PROGRAM LASER_PROG
VAR
	
	PULS1: TON;
	PULS2: TON;
	CNT1: CTU;
	LOTBOX_ACC: INT;
	LOTBOX_ACC1: INT;
	LOTBOX_TEMP1: INT;
	LOTBOX_TEMP2: INT;
	LOTBOX_TEMP3: INT;
	LOTBOX_TEMP4: INT;
	NGBOX_TEMP: INT;
	NGBOX_TEMP1: INT;
	NGBOX_TEMP2: INT;
	NGBOX_TEMP3: INT;
	NGBOX_TEMP4: INT;
	NGBOX_ACC: INT;
END_VAR


PULS1(IN:=NOT PULS2.Q,PT:=T#0.5S);
PULS2(IN:=PULS1.Q,PT:=T#1S);
CNT1(CU:=PULS1.Q,RESET:=CNT1.Q,PV:=9);
(*
IF CNT1.CV=1 THEN
	SORTER_VAR.O_NG_BOX_INDICATOR_4:=TRUE;
END_IF
IF CNT1.CV=2 THEN
	SORTER_VAR.O_NG_BOX_INDICATOR_3:=TRUE;
END_IF
IF CNT1.CV=3 THEN
	SORTER_VAR.O_NG_BOX_INDICATOR_2:=TRUE;
END_IF
IF CNT1.CV=4 THEN
	SORTER_VAR.O_NG_BOX_INDICATOR_1:=TRUE;
END_IF
IF CNT1.CV=5 THEN
	SORTER_VAR.O_LOT_BOX_INDICATOR_4:=TRUE;
END_IF
IF CNT1.CV=6 THEN
	SORTER_VAR.O_LOT_BOX_INDICATOR_3:=TRUE;
END_IF
IF CNT1.CV=7 THEN
	SORTER_VAR.O_LOT_BOX_INDICATOR_2:=TRUE;
END_IF
IF CNT1.CV=8 THEN
	SORTER_VAR.O_LOT_BOX_INDICATOR_1:=TRUE;
END_IF
IF CNT1.Q THEN
	SORTER_VAR.O_LOT_BOX_INDICATOR_1:=FALSE;
	SORTER_VAR.O_LOT_BOX_INDICATOR_2:=FALSE;
	SORTER_VAR.O_LOT_BOX_INDICATOR_3:=FALSE;
	SORTER_VAR.O_LOT_BOX_INDICATOR_4:=FALSE;
	SORTER_VAR.O_NG_BOX_INDICATOR_1:=FALSE;
	SORTER_VAR.O_NG_BOX_INDICATOR_2:=FALSE;
	SORTER_VAR.O_NG_BOX_INDICATOR_3:=FALSE;
	SORTER_VAR.O_NG_BOX_INDICATOR_4:=FALSE;
END_IF
*)
IF SORTER_VAR.I_LOTBOX_DETECT_1 THEN
	SORTER_VAR.O_LOT_BOX_INDICATOR_1:=PULS1.Q;
	LOTBOX_TEMP1:=1;
ELSE
	SORTER_VAR.O_LOT_BOX_INDICATOR_1:=FALSE;
	LOTBOX_TEMP1:=0;
END_IF

IF SORTER_VAR.I_LOTBOX_DETECT_2 THEN
	SORTER_VAR.O_LOT_BOX_INDICATOR_2:=PULS1.Q;
	LOTBOX_TEMP2:=1;
	ELSE
	LOTBOX_TEMP2:=0;
	SORTER_VAR.O_LOT_BOX_INDICATOR_2:=FALSE;
END_IF

IF SORTER_VAR.I_LOTBOX_DETECT_3 THEN
	SORTER_VAR.O_LOT_BOX_INDICATOR_3:=PULS1.Q;
	LOTBOX_TEMP3:=1;
	ELSE
	SORTER_VAR.O_LOT_BOX_INDICATOR_3:=FALSE;
	LOTBOX_TEMP3:=0;
END_IF

IF SORTER_VAR.I_LOTBOX_DETECT_4 THEN
	SORTER_VAR.O_LOT_BOX_INDICATOR_4:=PULS1.Q;
	LOTBOX_TEMP4:=1;
	ELSE
	SORTER_VAR.O_LOT_BOX_INDICATOR_4:=FALSE;
	LOTBOX_TEMP4:=0;
END_IF
LOTBOX_ACC:=LOTBOX_TEMP1 +LOTBOX_TEMP2+LOTBOX_TEMP3+LOTBOX_TEMP4;

IF LOTBOX_ACC >=3 THEN
	//SORTER_VAR.O_TOWER_LAMP_BUZZER :=TRUE;
	ELSE
	SORTER_VAR.O_TOWER_LAMP_BUZZER :=FALSE;
END_IF

IF NOT SORTER_VAR.I_NG_BOX_DETECT_1 THEN
		SORTER_VAR.O_NG_BOX_INDICATOR_1:=PULS1.Q;
		NGBOX_TEMP1:=1;
		ELSE
		SORTER_VAR.O_NG_BOX_INDICATOR_1:=FALSE;
		NGBOX_TEMP1:=0;
END_IF

IF NOT SORTER_VAR.I_NG_BOX_DETECT_2 THEN
		SORTER_VAR.O_NG_BOX_INDICATOR_2:=PULS1.Q;
		NGBOX_TEMP2:=1;
		ELSE
		SORTER_VAR.O_NG_BOX_INDICATOR_2:=FALSE;
		NGBOX_TEMP2:=0;
END_IF

IF NOT SORTER_VAR.I_NG_BOX_DETECT_3 THEN
		SORTER_VAR.O_NG_BOX_INDICATOR_3:=PULS1.Q;
		NGBOX_TEMP3:=1;
		ELSE
		SORTER_VAR.O_NG_BOX_INDICATOR_3:=FALSE;
		NGBOX_TEMP3:=0;
END_IF

IF NOT SORTER_VAR.I_NG_BOX_DETECT_4 THEN
		SORTER_VAR.O_NG_BOX_INDICATOR_4:=PULS1.Q;
		NGBOX_TEMP4:=1;
		ELSE
		SORTER_VAR.O_NG_BOX_INDICATOR_4:=FALSE;
		NGBOX_TEMP4:=0;
END_IF
NGBOX_ACC:=NGBOX_TEMP1+NGBOX_TEMP2+NGBOX_TEMP3+NGBOX_TEMP4;
IF NGBOX_ACC >=3 THEN
	//SORTER_VAR.O_TOWER_LAMP_BUZZER :=TRUE;
	ELSE
	SORTER_VAR.O_TOWER_LAMP_BUZZER :=FALSE;
END_IF

END_PROGRAM

(* stored: Version 1.1.0.1, ProductVersion 3.1.4020.12
   POU LASER_PROG: Id {75fe02f6-a49e-4e26-8a2d-398290aedd0e}, SpecialFunc None *)
